FUNCTION F_LeakMonitor_LUT_1 : FB_LeakMonitor
VAR_INPUT
END_VAR
VAR_OUTPUT
	// Provide stBoundaries output so test functions can reuse the boundaries
	stBoundaries : ST_LeakBoundaries := F_LeakBoundaries();
END_VAR
VAR
	fbLeakMonitor : FB_LeakMonitor;
END_VAR

fbLeakMonitor(
	bLeakDetected := TRUE,
	nLocationResistance := stBoundaries.nLMax5 -1,
	stBoundaries := stBoundaries
);

F_LeakMonitor_LUT_1 := fbLeakMonitor;

END_FUNCTION

(* stored: Version 1.1.0.1, ProductVersion 3.1.4020.14
   POU F_LeakMonitor_LUT_1: Id {29a3d80d-8d32-459d-84b9-1b050a987c74}, SpecialFunc None *)
